// TIA Portal V16 export
// export: Created 2022-02-28T20:45:44.7125792Z, ExportSetting WithDefaults, DisplayName Totally Integrated Automation Portal, DisplayVersion V16, DisplayName TIA Portal Version Control Interface, DisplayVersion V16, DisplayName TIA Portal Openness, DisplayVersion V16, DisplayName STEP 7 Professional, DisplayVersion V16, DisplayName STEP 7 Safety, DisplayVersion V16, DisplayName WinCC Advanced, DisplayVersion V16
FUNCTION "03_General" : Void   // FC3, LAD
{ S7_Optimized_Access := 'TRUE' }
VERSION : 0.1
// stored: AutoNumber true, IsIECCheckEnabled false, SetENOAutomatically false, UDAEnableTagReadback false
BEGIN

REGION Network 1: Confirmación Perifericos Pistilos
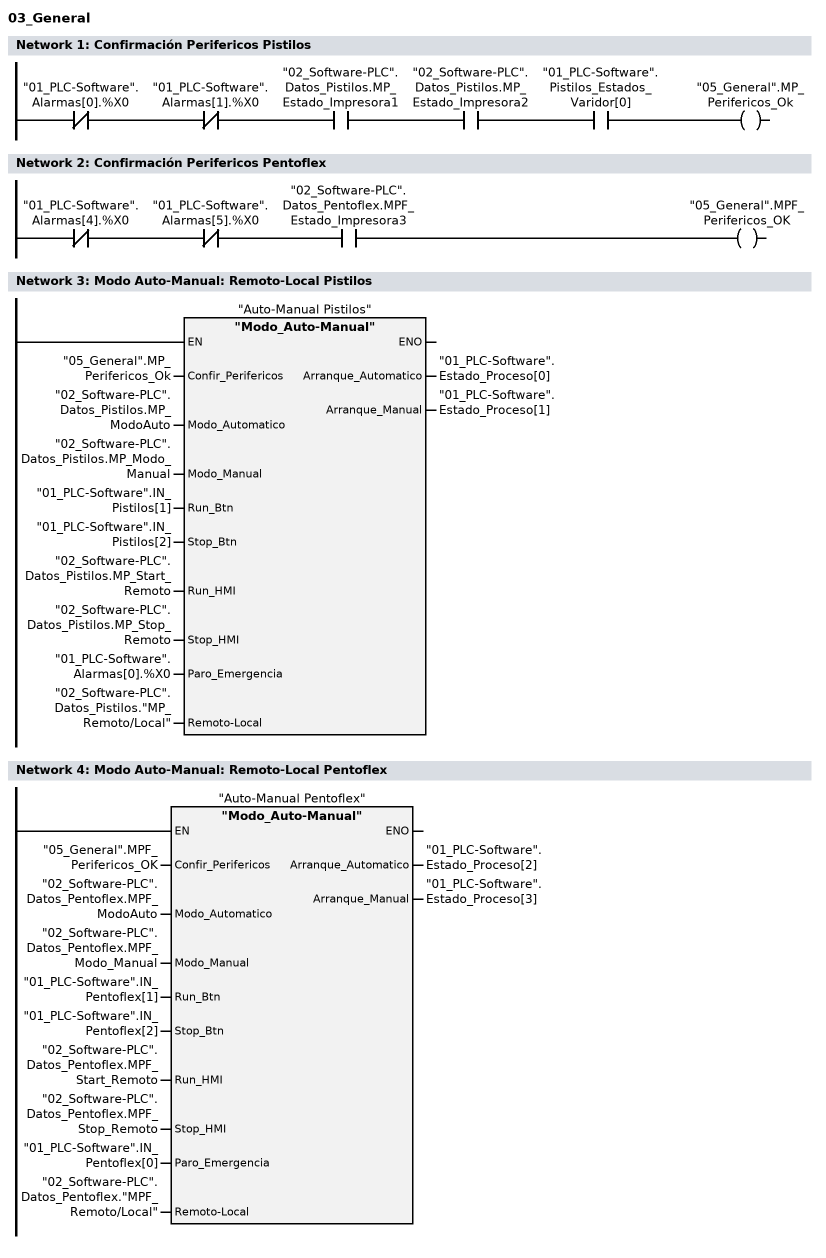
   RUNG wire#powerrail
      I_Contact( "01_PLC-Software".Alarmas[0].%X0 )
      I_Contact( "01_PLC-Software".Alarmas[1].%X0 )
      Contact( "02_Software-PLC".Datos_Pistilos.MP_Estado_Impresora1 )
      Contact( "02_Software-PLC".Datos_Pistilos.MP_Estado_Impresora2 )
      Contact( "01_PLC-Software".Pistilos_Estados_Varidor[0] )
      Coil( "05_General".MP_Perifericos_Ok )
   END_RUNG
   // the same network as SCL:
   "05_General".MP_Perifericos_Ok := NOT "01_PLC-Software".Alarmas[0].%X0 AND NOT "01_PLC-Software".Alarmas[1].%X0 AND "02_Software-PLC".Datos_Pistilos.MP_Estado_Impresora1 AND "02_Software-PLC".Datos_Pistilos.MP_Estado_Impresora2 AND "01_PLC-Software".Pistilos_Estados_Varidor[0];
END_REGION

REGION Network 2: Confirmación Perifericos Pentoflex
   RUNG wire#powerrail
      I_Contact( "01_PLC-Software".Alarmas[4].%X0 )
      I_Contact( "01_PLC-Software".Alarmas[5].%X0 )
      Contact( "02_Software-PLC".Datos_Pentoflex.MPF_Estado_Impresora3 )
      Coil( "05_General".MPF_Perifericos_OK )
   END_RUNG
   // the same network as SCL:
   "05_General".MPF_Perifericos_OK := NOT "01_PLC-Software".Alarmas[4].%X0 AND NOT "01_PLC-Software".Alarmas[5].%X0 AND "02_Software-PLC".Datos_Pentoflex.MPF_Estado_Impresora3;
END_REGION

REGION Network 3: Modo Auto-Manual: Remoto-Local Pistilos
   RUNG wire#powerrail
      "Auto-Manual Pistilos"(Confir_Perifericos := "05_General".MP_Perifericos_Ok, Modo_Automatico := "02_Software-PLC".Datos_Pistilos.MP_ModoAuto, Modo_Manual := "02_Software-PLC".Datos_Pistilos.MP_Modo_Manual, Run_Btn := "01_PLC-Software".IN_Pistilos[1], Stop_Btn := "01_PLC-Software".IN_Pistilos[2], Run_HMI := "02_Software-PLC".Datos_Pistilos.MP_Start_Remoto, Stop_HMI := "02_Software-PLC".Datos_Pistilos.MP_Stop_Remoto, Paro_Emergencia := "01_PLC-Software".Alarmas[0].%X0, "Remoto-Local" := "02_Software-PLC".Datos_Pistilos."MP_Remoto/Local", Arranque_Automatico => "01_PLC-Software".Estado_Proceso[0], Arranque_Manual => "01_PLC-Software".Estado_Proceso[1])
   END_RUNG
   // the same network as SCL:
   "Auto-Manual Pistilos"(Confir_Perifericos := "05_General".MP_Perifericos_Ok,   // "Modo_Auto-Manual"
                          Modo_Automatico := "02_Software-PLC".Datos_Pistilos.MP_ModoAuto,
                          Modo_Manual := "02_Software-PLC".Datos_Pistilos.MP_Modo_Manual,
                          Run_Btn := "01_PLC-Software".IN_Pistilos[1],
                          Stop_Btn := "01_PLC-Software".IN_Pistilos[2],
                          Run_HMI := "02_Software-PLC".Datos_Pistilos.MP_Start_Remoto,
                          Stop_HMI := "02_Software-PLC".Datos_Pistilos.MP_Stop_Remoto,
                          Paro_Emergencia := "01_PLC-Software".Alarmas[0].%X0,
                          "Remoto-Local" := "02_Software-PLC".Datos_Pistilos."MP_Remoto/Local",
                          Arranque_Automatico => "01_PLC-Software".Estado_Proceso[0],
                          Arranque_Manual => "01_PLC-Software".Estado_Proceso[1]);
END_REGION

REGION Network 4: Modo Auto-Manual: Remoto-Local Pentoflex
   RUNG wire#powerrail
      "Auto-Manual Pentoflex"(Confir_Perifericos := "05_General".MPF_Perifericos_OK, Modo_Automatico := "02_Software-PLC".Datos_Pentoflex.MPF_ModoAuto, Modo_Manual := "02_Software-PLC".Datos_Pentoflex.MPF_Modo_Manual, Run_Btn := "01_PLC-Software".IN_Pentoflex[1], Stop_Btn := "01_PLC-Software".IN_Pentoflex[2], Run_HMI := "02_Software-PLC".Datos_Pentoflex.MPF_Start_Remoto, Stop_HMI := "02_Software-PLC".Datos_Pentoflex.MPF_Stop_Remoto, Paro_Emergencia := "01_PLC-Software".IN_Pentoflex[0], "Remoto-Local" := "02_Software-PLC".Datos_Pentoflex."MPF_Remoto/Local", Arranque_Automatico => "01_PLC-Software".Estado_Proceso[2], Arranque_Manual => "01_PLC-Software".Estado_Proceso[3])
   END_RUNG
   // the same network as SCL:
   "Auto-Manual Pentoflex"(Confir_Perifericos := "05_General".MPF_Perifericos_OK,   // "Modo_Auto-Manual"
                           Modo_Automatico := "02_Software-PLC".Datos_Pentoflex.MPF_ModoAuto,
                           Modo_Manual := "02_Software-PLC".Datos_Pentoflex.MPF_Modo_Manual,
                           Run_Btn := "01_PLC-Software".IN_Pentoflex[1],
                           Stop_Btn := "01_PLC-Software".IN_Pentoflex[2],
                           Run_HMI := "02_Software-PLC".Datos_Pentoflex.MPF_Start_Remoto,
                           Stop_HMI := "02_Software-PLC".Datos_Pentoflex.MPF_Stop_Remoto,
                           Paro_Emergencia := "01_PLC-Software".IN_Pentoflex[0],
                           "Remoto-Local" := "02_Software-PLC".Datos_Pentoflex."MPF_Remoto/Local",
                           Arranque_Automatico => "01_PLC-Software".Estado_Proceso[2],
                           Arranque_Manual => "01_PLC-Software".Estado_Proceso[3]);
END_REGION
END_FUNCTION
